TEXTLIST GroupState_txt
  0 = 'INVALID'
  1 = 'DISABLED'
  2 = 'STANDBY'
  3 = 'MOVING'
  4 = 'STOPPING'
  5 = 'ERROR STOP'
  6 = 'HOMING'
  7 = 'NOT READY'
  8 = 'SUSPENDED'
   = ''
END_TEXTLIST

(* stored: Version 1.1.0.1, ProductVersion 3.1.4024.11
   TextList GroupState_txt: Id {80b17d88-9834-4c7d-a12d-076eaf4fe542} *)
